RoboDK station: crx10_demo.rdk

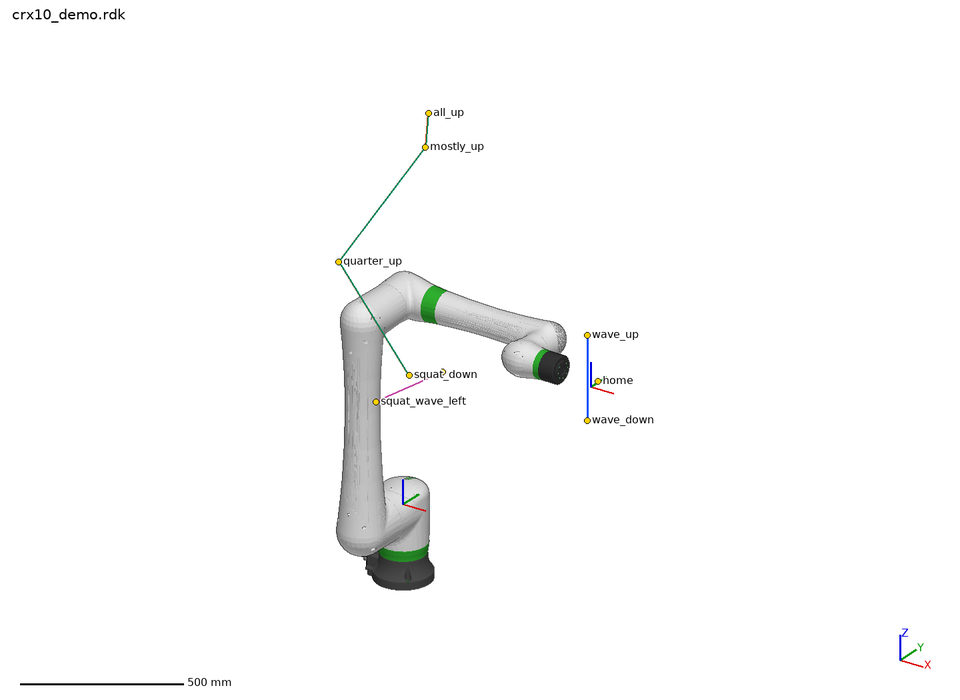
[picture v0: the station drawn from its stored meshes, robots at their saved joint values, targets as dots, program paths as lines]
Station crx10_demo (saved by RoboDK 5.5.4). Poses are relative to the parent item; angles as X-Y-Z fixed-axis rotations.
Station parameters (name, value as stored): LIN64
  - frame Fanuc CRX-10iA/L Base at (0, 0, 245) mm
    - robot Fanuc CRX-10iA/L: 6 axes, payload 10 kg, reach 1418 mm, repeatability 0.05 mm, weight 40 kg
        modified DH rows (alpha deg, a mm, theta deg, d mm): 0, 0, 0, 245; -90, 0, -90, 0; 0, 710, 0, 0; -90, 0, 0, 540; 90, 0, 0, -150; -90, 0, 0, 160
        base shift (0, 0, -245) mm
        joint limits [-180, -180, -360, -190, -180, -190] to [180, 180, 430, 190, 180, 190]; home [0, 0, 0, 0, 0, 0]; saved at [0, 0, 0, 0, 0, 0]
      - tool RobotiQ 2F-85 Gripper (Open), TCP at (0, 0, 130) mm, size 147.4 x 75 x 146.8 mm
    - frame refPoint at (0, 1000, 0) mm
      - target squat_down (Cartesian target) at (127.18, -1150, 532.83) mm, rotated rx 0 ry 0 rz -180 deg; joints [80.588, -70, 0, 0, 90, 80.588] of Fanuc CRX-10iA/L
      - target quarter_up (Cartesian target) at (-161.59, -1111.99, 822.61) mm, rotated rx -0.01 ry 0 rz -104.23 deg; joints [-15, -62.21, 21.92, 0, 68.07, -90.773] of Fanuc CRX-10iA/L
      - target mostly_up (Cartesian target) at (-50.05, -809.96, 1122.8) mm, rotated rx 0.02 ry -0.01 rz -15 deg; joints [-125, -48.24, 41.8, 0, 48.18, 70] of Fanuc CRX-10iA/L
      - target all_up (Cartesian target) at (166.83, -1103.35, 1415.83) mm, rotated rx -0.01 ry 0.03 rz 98.44 deg; joints [-162, -28, 67.49, 179.92, -22.5, 99.63] of Fanuc CRX-10iA/L
      - target home (Cartesian target) at (830, -1150, 710) mm, rotated rx 0 ry -90 rz -180 deg; joints [0, 0, 0, 0, 0, 0] of Fanuc CRX-10iA/L
      - target wave_down (Cartesian target) at (791.15, -1150, 565) mm, rotated rx -180 ry -60 rz 0 deg; joints [0, 0, 0, 0, -30, 0] of Fanuc CRX-10iA/L
      - target wave_up (Cartesian target) at (791.15, -1150, 855) mm, rotated rx 0 ry -60 rz -180 deg; joints [0, 0, 0, 0, 30, 0] of Fanuc CRX-10iA/L
      - target squat_wave_right (Cartesian target) at (150.89, -1006.95, 493.98) mm, rotated rx 29.67 ry -4.69 rz 178.76 deg; joints [80.59, -70, 0, 0, 60, 80.59] of Fanuc CRX-10iA/L
      - target squat_wave_left (Cartesian target) at (103.48, -1293.04, 493.98) mm, rotated rx -29.67 ry 4.69 rz 178.76 deg; joints [80.59, -70, 0, 0, 120, 80.59] of Fanuc CRX-10iA/L
  - program wave (6 instructions, listed below)
  - program spin_up (6 instructions, listed below)
  - program spin_down (6 instructions, listed below)
  - program squat_wave (6 instructions, listed below)
  - program main (5 instructions, listed below)
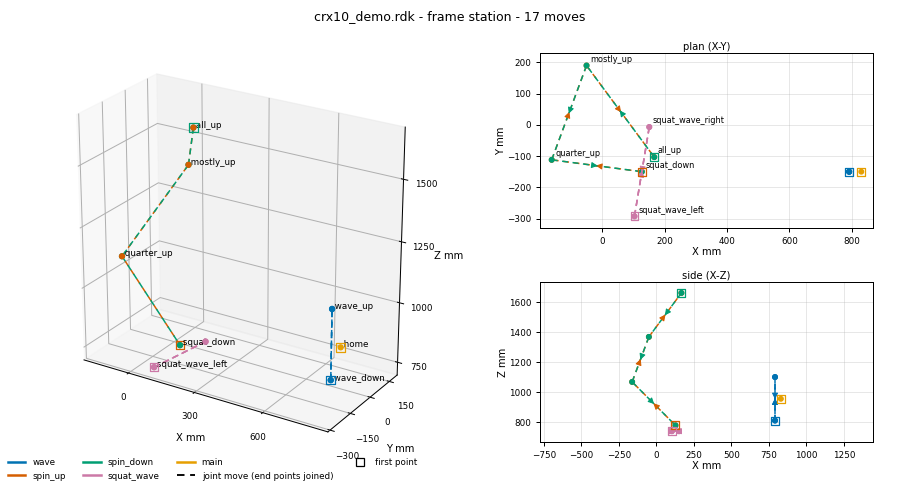
[picture p0: tool path of crx10_demo.rdk in frame station, 17 of 17 moves have a stored position in this frame; points joined in program order, loops and branches not executed]

--- program wave (robot Fanuc CRX-10iA/L) ---
  Set Ref.: refPoint
  Set Tool: RobotiQ 2F-85 Gripper (Open)
  MoveJ (wave_down)
  MoveJ (wave_up)
  MoveJ (wave_down)
  MoveJ (wave_up)

--- program spin_up (robot Fanuc CRX-10iA/L) ---
  Set Ref.: refPoint
  Set Tool: RobotiQ 2F-85 Gripper (Open)
  MoveJ (squat_down)
  MoveJ (quarter_up)
  MoveJ (mostly_up)
  MoveJ (all_up)

--- program spin_down (robot Fanuc CRX-10iA/L) ---
  Set Ref.: refPoint
  Set Tool: RobotiQ 2F-85 Gripper (Open)
  MoveJ (all_up)
  MoveJ (mostly_up)
  MoveJ (quarter_up)
  MoveJ (squat_down)

--- program squat_wave (robot Fanuc CRX-10iA/L) ---
  Set Ref.: refPoint
  Set Tool: RobotiQ 2F-85 Gripper (Open)
  MoveJ (squat_wave_left)
  MoveJ (squat_wave_right)
  MoveJ (squat_wave_left)
  MoveJ (squat_wave_right)

--- program main (robot Fanuc CRX-10iA/L) ---
  Call wave
  Call spin_up
  Call spin_down
  Call squat_wave
  MoveJ (home)
